ADAPTER ADP_ORDER_DATA (* Adapter Interface *)
  (* Standard: 61499-1 *)
  (* Version 0.0, 12/17/2022, Dmitrii, Flexbridge AB *)
  PACKAGE UAO.Hackathon;
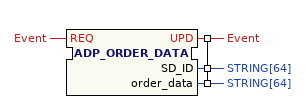
  EVENT_INPUT
    REQ;
  END_EVENT
  EVENT_OUTPUT
    UPD WITH SD_ID, order_data; (* Confirmation from Plug *)
  END_EVENT
  VAR_OUTPUT
    SD_ID : STRING[64]; (* Confirmation Data from Plug *)
    order_data : STRING[64]; (* Indication Data from Plug *)
  END_VAR
  SERVICE SOCKET/PLUG
    SEQUENCE request_confirm
      SOCKET.UPD(REQD) -> PLUG.UPD(REQD);
      PLUG.UPD(SD_ID) -> SOCKET.UPD(SD_ID);
    END_SEQUENCE
    SEQUENCE indication_response
      PLUG.IND(order_data) -> SOCKET.IND(order_data);
      SOCKET.RSP(RSPD) -> PLUG.RSP(RSPD);
    END_SEQUENCE
  END_SERVICE
END_ADAPTER
